TYPE ST_Tank :
STRUCT
	id : INT;
	temperature : REAL:=93;
	level : REAL:=94;
	alarm : BOOL;
END_STRUCT
END_TYPE

(* stored: Version 1.1.0.1, ProductVersion 3.1.4024.16
   DUT ST_Tank: Id {e0ddc1ad-9b37-4cdd-b6a7-a91f6c3597f9} *)
